{attribute 'linkalways'} 
{attribute 'no_explicit_call' := 'This FB is a CLASS and must be accessed using methods or properties'}
{attribute 'enable_dynamic_creation'}
FUNCTION_BLOCK Node_F_VN_ContourPerimeter EXTENDS VisionNode
VAR
    ipContour : _ITcVnContainer;
    fPerimeter : _LREAL(0.0);
    bClosed : _BOOL(FALSE);
    hrPrev : _HRESULT(S_OK);
	hresult : _HRESULT(S_OK);
END_VAR

METHOD PUBLIC  Clone : I_Node
VAR
	pNode : POINTER TO Node_F_VN_ContourPerimeter;
END_VAR
pNode := __NEW(Node_F_VN_ContourPerimeter);
Clone := pNode^;
END_METHOD

METHOD FB_init : BOOL
VAR_INPUT
	bInitRetains : BOOL; // if TRUE, the retain variables are initialized (warm start / cold start)
	bInCopyCode : BOOL;  // if TRUE, the instance afterwards gets moved into the copy code (online change)
END_VAR
AddInput('ipContour', ipContour);
AddParameter('bClosed', bClosed);
AddInput('hrPrev', hrPrev);
AddOutput('fPerimeter', fPerimeter);
AddOutput('hresult',hresult);
END_METHOD

METHOD PROTECTED OnExecute
hresult.Value := F_VN_ContourPerimeter(
	ipContour := ipContour.Value,
    fPerimeter := fPerimeter.Value,
    bClosed := bClosed.Value,
	hrPrev:= hrPrev.Value);
END_METHOD

METHOD PUBLIC PreExecutionCheck
VAR_INPUT
	Check : I_PreExecutionChecks;
END_VAR
Check.IsTrue(ipContour.IsValid, 'ipContour must be a valid container');
Check.IsTrue((ipContour.IsType(TC_GLOBAL_CONST_LIST.ContainerType_Vector_TcVnPoint2_DINT) OR
              ipContour.IsType(TC_GLOBAL_CONST_LIST.ContainerType_Vector_TcVnPoint2_REAL)),
              'ipContour contains incorrect type');
END_METHOD

END_FUNCTION_BLOCK

(* stored: Version 1.1.0.1, ProductVersion 3.1.4026.13
   POU Node_F_VN_ContourPerimeter: Id {2c8d2e9c-d541-0922-177d-7597bc293858}, SpecialFunc None
   Folder Constructor: Id {bbca1b00-dd39-084a-2a5a-50ce3d89cc76}
   Method Clone: Id {da7539dd-35df-0e60-29f5-6ab0e239b3c0}
   Method FB_init: Id {f116b094-2671-0c8a-1662-1e32438751b4}
   Method OnExecute: Id {476f953a-2602-0df7-234a-42ee0a323dbc}
   Method PreExecutionCheck: Id {3ccdf60f-1520-0791-1b94-bc87bf361f3c} *)
